FUNCTION_BLOCK FB_TEST2
VAR_INPUT
	execute: BOOL;
	pos2: LREAL := 2500;
END_VAR
VAR
	TIMERDONE: BOOL;
END_VAR

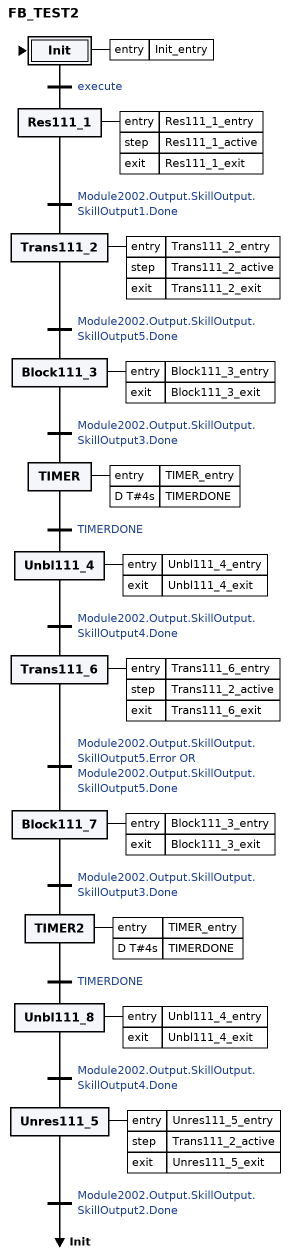
INITIAL_STEP Init:
    Init_entry(P1);  // entry action
END_STEP
TRANSITION FROM Init TO Res111_1
    := execute;
END_TRANSITION
STEP Res111_1:
    Res111_1_entry(P1);  // entry action
    Res111_1_active(N);  // step action
    Res111_1_exit(P0);  // exit action
END_STEP
TRANSITION FROM Res111_1 TO Trans111_2
    := Module2002.Output.SkillOutput.SkillOutput1.Done;
END_TRANSITION
STEP Trans111_2:
    Trans111_2_entry(P1);  // entry action
    Trans111_2_active(N);  // step action
    Trans111_2_exit(P0);  // exit action
END_STEP
TRANSITION FROM Trans111_2 TO Block111_3
    := Module2002.Output.SkillOutput.SkillOutput5.Done;
END_TRANSITION
STEP Block111_3:
    Block111_3_entry(P1);  // entry action
    Block111_3_exit(P0);  // exit action
END_STEP
TRANSITION FROM Block111_3 TO TIMER
    := Module2002.Output.SkillOutput.SkillOutput3.Done;
END_TRANSITION
STEP TIMER:
    TIMER_entry(P1);  // entry action
    TIMERDONE(D, T#4s);
END_STEP
TRANSITION FROM TIMER TO Unbl111_4
    := TIMERDONE;
END_TRANSITION
STEP Unbl111_4:
    Unbl111_4_entry(P1);  // entry action
    Unbl111_4_exit(P0);  // exit action
END_STEP
TRANSITION FROM Unbl111_4 TO Trans111_6
    := Module2002.Output.SkillOutput.SkillOutput4.Done;
END_TRANSITION
STEP Trans111_6:
    Trans111_6_entry(P1);  // entry action
    Trans111_2_active(N);  // step action
    Trans111_6_exit(P0);  // exit action
END_STEP
TRANSITION FROM Trans111_6 TO Block111_7
    := Module2002.Output.SkillOutput.SkillOutput5.Error OR Module2002.Output.SkillOutput.SkillOutput5.Done;
END_TRANSITION
STEP Block111_7:
    Block111_3_entry(P1);  // entry action
    Block111_3_exit(P0);  // exit action
END_STEP
TRANSITION FROM Block111_7 TO TIMER2
    := Module2002.Output.SkillOutput.SkillOutput3.Done;
END_TRANSITION
STEP TIMER2:
    TIMER_entry(P1);  // entry action
    TIMERDONE(D, T#4s);
END_STEP
TRANSITION FROM TIMER2 TO Unbl111_8
    := TIMERDONE;
END_TRANSITION
STEP Unbl111_8:
    Unbl111_4_entry(P1);  // entry action
    Unbl111_4_exit(P0);  // exit action
END_STEP
TRANSITION FROM Unbl111_8 TO Unres111_5
    := Module2002.Output.SkillOutput.SkillOutput4.Done;
END_TRANSITION
STEP Unres111_5:
    Unres111_5_entry(P1);  // entry action
    Trans111_2_active(N);  // step action
    Unres111_5_exit(P0);  // exit action
END_STEP
TRANSITION FROM Unres111_5 TO Init
    := Module2002.Output.SkillOutput.SkillOutput2.Done;
END_TRANSITION

ACTION Trans111_6_exit:
//TRANSPORTIEREN

Module2002.Input.SkillInput.SkillInput5.Execute := FALSE;
Module2002.Input.SkillInput.SkillInput5.ParameterInput.Parameterinput1.Value := 0; //X-Position
Module2002.Input.SkillInput.SkillInput5.ParameterInput.Parameterinput2.Value := 0; //Z-Position
Module2002.Input.SkillInput.SkillInput5.ParameterInput.Parameterinput3.Value := 0; //Velocity
Module2002.Input.SkillInput.SkillInput5.ParameterInput.Parameterinput4.Value := 0; //Acceleration
END_ACTION

ACTION Block111_3_entry:
//BLOCKIEREN

Module2002.Input.SkillInput.SkillInput3.Execute := TRUE;
Module2002.Input.SkillInput.SkillInput3.ParameterInput.Parameterinput1.Value := 112; //TaskID
END_ACTION

ACTION Trans111_6_entry:
//TRANSPORTIEREN

Module2002.Input.SkillInput.SkillInput5.Execute := TRUE;
Module2002.Input.SkillInput.SkillInput5.ParameterInput.Parameterinput1.Value := pos2; //X-Position
Module2002.Input.SkillInput.SkillInput5.ParameterInput.Parameterinput2.Value := 80; //Z-Position
Module2002.Input.SkillInput.SkillInput5.ParameterInput.Parameterinput3.Value := 0; //Velocity
Module2002.Input.SkillInput.SkillInput5.ParameterInput.Parameterinput4.Value := 0; //Acceleration
END_ACTION

ACTION Init_entry:
execute := FALSE;
END_ACTION

ACTION Trans111_2_entry:
//TRANSPORTIEREN

Module2002.Input.SkillInput.SkillInput5.Execute := TRUE;
Module2002.Input.SkillInput.SkillInput5.ParameterInput.Parameterinput1.Value := 3000; //X-Position
Module2002.Input.SkillInput.SkillInput5.ParameterInput.Parameterinput2.Value := 0; //Z-Position
Module2002.Input.SkillInput.SkillInput5.ParameterInput.Parameterinput3.Value := 0; //Velocity
Module2002.Input.SkillInput.SkillInput5.ParameterInput.Parameterinput4.Value := 0; //Acceleration
END_ACTION

ACTION Res111_1_entry:
// Reservieren entry
Module2002.Input.SkillInput.SkillInput1.Execute := TRUE;
Module2002.Input.SkillInput.SkillInput1.ParameterInput.Parameterinput1.Value := 112; //TASKID
END_ACTION

ACTION Unbl111_4_exit:
//unBLOCKIEREN

Module2002.Input.SkillInput.SkillInput4.Execute := FALSE; 
Module2002.Input.SkillInput.SkillInput4.ParameterInput.Parameterinput1.Value := 000; //TaskID
END_ACTION

ACTION Unres111_5_entry:
//unreserve
Module2002.Input.SkillInput.SkillInput2.Execute := TRUE;
Module2002.Input.SkillInput.SkillInput2.ParameterInput.Parameterinput1.Value := 112; //TaskID
END_ACTION

ACTION Res111_1_active:

END_ACTION

ACTION Trans111_2_exit:
//TRANSPORTIEREN

Module2002.Input.SkillInput.SkillInput5.Execute := FALSE;
Module2002.Input.SkillInput.SkillInput5.ParameterInput.Parameterinput1.Value := 0; //X-Position
Module2002.Input.SkillInput.SkillInput5.ParameterInput.Parameterinput2.Value := 0; //Z-Position
Module2002.Input.SkillInput.SkillInput5.ParameterInput.Parameterinput3.Value := 0; //Velocity
Module2002.Input.SkillInput.SkillInput5.ParameterInput.Parameterinput4.Value := 0; //Acceleration
END_ACTION

ACTION TIMER_entry:
TIMERDONE := FALSE;
END_ACTION

ACTION Trans111_2_active:

END_ACTION

ACTION Unbl111_4_entry:
//unBLOCKIEREN

Module2002.Input.SkillInput.SkillInput4.Execute := TRUE; //FALSE weil timer
Module2002.Input.SkillInput.SkillInput4.ParameterInput.Parameterinput1.Value := 112; //TaskID
END_ACTION

ACTION Trans111_2_entry_1:
//TRANSPORTIEREN

Module2002.Input.SkillInput.SkillInput5.Execute := TRUE;
Module2002.Input.SkillInput.SkillInput5.ParameterInput.Parameterinput1.Value := 3000; //X-Position
Module2002.Input.SkillInput.SkillInput5.ParameterInput.Parameterinput2.Value := 0; //Z-Position
Module2002.Input.SkillInput.SkillInput5.ParameterInput.Parameterinput3.Value := 0; //Velocity
Module2002.Input.SkillInput.SkillInput5.ParameterInput.Parameterinput4.Value := 0; //Acceleration
END_ACTION

ACTION Unres111_5_exit:
//unreserve
Module2002.Input.SkillInput.SkillInput2.Execute := FALSE;
Module2002.Input.SkillInput.SkillInput2.ParameterInput.Parameterinput1.Value := 0; //TaskID
END_ACTION

ACTION Block111_3_exit:
//BLOCKIEREN

Module2002.Input.SkillInput.SkillInput3.Execute := FALSE;
Module2002.Input.SkillInput.SkillInput3.ParameterInput.Parameterinput1.Value := 0; //TaskID
END_ACTION

ACTION Res111_1_exit:
// Reservieren entry
Module2002.Input.SkillInput.SkillInput1.Execute := FALSE;
Module2002.Input.SkillInput.SkillInput1.ParameterInput.Parameterinput1.Value := 0; //TASKID
END_ACTION

END_FUNCTION_BLOCK

(* stored: Version 1.1.0.1, ProductVersion 3.1.0.25
   POU FB_TEST2: Id {9d4b7242-75b0-4d4b-bb68-6e5c4eaa7530}
   Action Trans111_6_exit: Id {11f3b906-8180-4057-967a-5b9d0a7caa17}
   Action Block111_3_entry: Id {1db0218d-5c6e-49e6-9c35-d4f1b9dfc5e9}
   Action Trans111_6_entry: Id {22dc55d4-2554-4e50-ba3c-2d69eee09a9c}
   Action Init_entry: Id {4f1609ba-7ad3-41e4-a0d4-1adba173f851}
   Action Trans111_2_entry: Id {5ced6d16-f543-4844-b8b3-705fb5814283}
   Action Res111_1_entry: Id {785dff91-1d5f-4029-8aa8-5589bece6624}
   Action Unbl111_4_exit: Id {7c06ddff-b426-4084-9b57-c4008a636fa3}
   Action Unres111_5_entry: Id {9419857b-0a78-42f2-9ec2-4c8f0c5672f7}
   Action Res111_1_active: Id {989b894c-1cfc-492a-84eb-063769358ca7}
   Action Trans111_2_exit: Id {a01dcc76-ccad-4a8a-9d4e-363db9aa0b4b}
   Action TIMER_entry: Id {a5a4587e-d994-4d42-b254-d58f46d53cf1}
   Action Trans111_2_active: Id {aa0c1763-e9dd-4934-a073-ee8c01c8a9c8}
   Action Unbl111_4_entry: Id {cfd719e7-ee95-4183-92ec-3dcebd89f1c9}
   Action Trans111_2_entry_1: Id {d0664484-a3a3-4f84-8c42-79ef9c2bf345}
   Action Unres111_5_exit: Id {dfb0634f-55ad-4954-84b2-46ad988d95cd}
   Action Block111_3_exit: Id {e78a9f06-4e8a-4cf0-a194-67dbda45dede}
   Action Res111_1_exit: Id {f6a833c4-a2c2-4512-be5f-eda5c5366529} *)
